PROGRAM MAIN
VAR

	fbMyPizzaOven : FB_PIZZA_OVEN;

	fbMyPizzaOven1 : FB_PIZZA_OVEN;
	
	bLoadPizza   : BOOL;
	bRemovePizza : BOOL;	
	
END_VAR



fbMyPizzaOven(bLoadPizza:= bLoadPizza, bRemovePizza:=bRemovePizza);


fbMyPizzaOven1(bLoadPizza:= bLoadPizza, bRemovePizza:=bRemovePizza);

END_PROGRAM

(* stored: Version 1.1.0.1, ProductVersion 3.1.4020.3
   POU MAIN: Id {f9a624a7-3b5f-4807-8bd7-72971c0fcf58}, SpecialFunc None *)
